FUNCTION_BLOCK FWKinematics
VAR_INPUT
	par : ST_pValveControlledCylinder;
	fbCraneAngle : CraneAngle;
	L1 : LREAL;
	L2 : LREAL;
	L3 : LREAL;
	L4 : LREAL;
	thetaSlew : LREAL;
	thetaMainBoom : LREAL;
	thetaKnuckleBoom : LREAL;
END_VAR
VAR_OUTPUT
	X : LREAL;
	Y : LREAL;
	Z : LREAL;
END_VAR
VAR
END_VAR






X := COS(thetaSlew)*(L2 + L4*COS(thetaMainBoom + thetaKnuckleBoom) + L3*COS(thetaMainBoom));
Y := SIN(thetaSlew)*(L2 + L4*COS(thetaMainBoom + thetaKnuckleBoom) + L3*COS(thetaMainBoom));
Z := L1 + L4*SIN(thetaMainBoom + thetaKnuckleBoom) + L3*SIN(thetaMainBoom);

END_FUNCTION_BLOCK

(* stored: Version 1.1.0.1, ProductVersion 3.1.4024.9
   POU FWKinematics: Id {7097862a-1caf-42f1-82d5-88fbe7cef7b9}, SpecialFunc None *)
